Universal Robots URScript: pieza_4_ur5_recoger.urscript

def ur5e_recoger_baldosa_simulada():
  textmsg("=== UR5e PARTE 1: recoger baldosa simulada ===")

  q_home = p[0.54216, -0.32723, 0.38191, 3.06600, -0.68500, 0.00000]

  # X/Y llegan DIRECTAMENTE del JSON. NO se corrige nada aquí.
  x_pick = 0.01171
  y_pick = -0.32762

  # Orientacion real medida en tablet para coger piezas.
  rx_pick = 2.79604
  ry_pick = -1.43234
  rz_pick = 0.00003

  # Orientacion propia de DROP_ZONE.
  rx_drop = 1.96260
  ry_drop = 2.48200
  rz_drop = 0.00000

  textmsg("UR5e TARGET JSON x=0.01171, y=-0.32762")
  textmsg("UR5e ORIENT PICK rx=2.79604, ry=-1.43234, rz=0.00003")
  textmsg("Angulo vision ignorado=-38.19")

  # 1) HOME -> punto alto justo encima de la pieza
  textmsg("UR5e: yendo a HOME")
  movej(q_home, a=0.03, v=0.1)
  sleep(0.3)
  movej(p[x_pick, y_pick, 0.25000, rx_pick, ry_pick, rz_pick], a=0.12, v=0.08)
  sleep(0.3)
  textmsg("UR5e pieza original: detectando superficie por fuerza")
  zero_ftsensor()
  sleep(0.5)
  i_f = 0
  while (force() < 1.500 and i_f < 8000):
    speedl([0, 0, -0.00800, 0, 0, 0], 0.15, 0.02)
    i_f = i_f + 1
  end
  stopl(2.0)
  sleep(0.2)
  if (i_f >= 8000):
    popup("UR5e pieza original: no se detecto contacto. Revisa posicion/Z/fuerza.", error=True)
    halt
  end
  z_contacto = get_actual_tcp_pose()[2]
  z_trabajo = z_contacto + 0.00300
  textmsg("UR5e pieza original: z_contacto=", z_contacto)
  textmsg("SIMULACION: ventosa ON / pieza cogida")
  sleep(0.40)

  # 2) Retirada por el mismo punto alto de entrada
  movel(p[x_pick, y_pick, 0.25000, rx_pick, ry_pick, rz_pick], a=0.03, v=0.08)
  sleep(0.2)
  textmsg("UR5e: yendo a HOME")
  movej(q_home, a=0.03, v=0.1)
  sleep(0.3)

  # 3) HOME -> DROP_ZONE
  movej(p[-0.04511, 0.51128, 0.29870, 1.96260, 2.48200, 0.00000], a=0.12, v=0.125)
  sleep(0.3)
  textmsg("UR5e deposito DROP_ZONE: detectando superficie por fuerza")
  zero_ftsensor()
  sleep(0.5)
  i_f = 0
  while (force() < 1.500 and i_f < 8000):
    speedl([0, 0, -0.00800, 0, 0, 0], 0.15, 0.02)
    i_f = i_f + 1
  end
  stopl(2.0)
  sleep(0.2)
  if (i_f >= 8000):
    popup("UR5e deposito DROP_ZONE: no se detecto contacto. Revisa posicion/Z/fuerza.", error=True)
    halt
  end
  z_contacto = get_actual_tcp_pose()[2]
  z_trabajo = z_contacto + 0.00300
  textmsg("UR5e deposito DROP_ZONE: z_contacto=", z_contacto)
  textmsg("SIMULACION: ventosa OFF / pieza soltada")
  sleep(0.30)

  # 4) Retirada por el mismo punto alto de DROP_ZONE
  movel(p[-0.04511, 0.51128, 0.29870, 1.96260, 2.48200, 0.00000], a=0.03, v=0.08)
  sleep(0.2)
  textmsg("UR5e: yendo a HOME")
  movej(q_home, a=0.03, v=0.1)
  sleep(0.3)

  textmsg("UR5e: baldosa simulada en DROP_ZONE. Avisando al PC")
  # === Aviso al PC: UR5e ===
  socket_ok = socket_open("192.168.56.2", 50001, "sync_ur5_ur3")
  if (not socket_ok):
    popup("UR5e: no pudo avisar al PC", error=True)
    halt
  else:
    socket_send_string("LISTO", "sync_ur5_ur3")
    sleep(0.2)
    socket_close("sync_ur5_ur3")
    textmsg("UR5e: LISTO enviado al PC")
  end
  textmsg("UR5e PARTE 1 finalizada")
end
ur5e_recoger_baldosa_simulada()
